// TIA Portal V20 export
// export: Created 2025-12-01T14:56:22.4264934Z, ExportSetting None, DisplayName Totally Integrated Automation Portal, DisplayVersion V20 Update 3, DisplayName TIA Portal Openness, DisplayVersion V20 Update 3, DisplayName TIA Portal Version Control Interface, DisplayVersion V20 Update 3, DisplayName STEP 7 Professional, DisplayVersion V20 Update 3, DisplayName STEP 7 Safety, DisplayVersion V20 Update 2, DisplayName WinCC Basic/Comfort/Advanced, DisplayVersion V20 Update 3, DisplayName WinCC Professional, DisplayVersion V20 Update 3, DisplayName WinCC Unified, DisplayVersion V20 Update 3
TYPE "UDT_MesaMaquina_Interlock"
   STRUCT
      CargaAct_Dcha : Bool;
      DesCargaAct_Dcha : Bool;
      AVTF_Dcha : Bool;
      P_Mens_Dcha : Bool;
      PTF_Dcha : Bool;
      FTF_Dcha : Bool;
      CargaAct_Izq : Bool;
      DesCargaAct_Izq : Bool;
      AVTF_Izq : Bool;
      P_Mens_Izq : Bool;
      PTF_Izq : Bool;
      FTF_Izq : Bool;
   END_STRUCT;
END_TYPE
